FUNCTION_BLOCK Fb_CalculoCoordenadasFinalesFormacion
VAR_INPUT
	TipoCalForCavallete 					: UINT ;
	numeroLastre_int 						: UINT ;
	TipoRisultato							: UINT ;
	AlgoloAlfa_gradi						: LREAL ;
	CalculoEstacionPickinPiezasDiferentes 	: BOOL ;
	Supporto 								: POINTER TO TFMachinePalletizer_Pallet;
	XFinale 								: POINTER TO  ARRAY [1..MAXFORMINGSLAB] OF LREAL;
	
	CoorFinaleLado_Pri0_Des180 : POINTER TO ARRAY [1..MAXFORMINGSLAB] OF Es_CoordenadasCaballeteLadoA_ladoB ;
	
	YFinale 					: POINTER TO  ARRAY [1..MAXFORMINGSLAB] OF LREAL;
	YInternoLastra 				: POINTER TO  ARRAY [1..MAXFORMINGSLAB] OF LREAL;
	YCentroLastra				: POINTER TO  ARRAY [1..MAXFORMINGSLAB] OF LREAL;
	YEsternoLastra				: POINTER TO  ARRAY [1..MAXFORMINGSLAB] OF LREAL;
	YCoordinataAppoggioLastra 	: POINTER TO  ARRAY [1..MAXFORMINGSLAB] OF LREAL;
	
	ZFinale 					: POINTER TO  ARRAY [1..MAXFORMINGSLAB] OF LREAL;
	ZInternoLastra				: POINTER TO  ARRAY [1..MAXFORMINGSLAB] OF LREAL;
	ZCentroLastra      			: POINTER TO  ARRAY [1..MAXFORMINGSLAB] OF LREAL;
	ZEsternoLastra				: POINTER TO  ARRAY [1..MAXFORMINGSLAB] OF LREAL;
	
	JFinale 					: POINTER TO  ARRAY [1..MAXFORMINGSLAB] OF LREAL;
	
	XInternoLastra_A_B : POINTER TO ARRAY [1..MAXFORMINGSLAB] OF ES_SpesoreLastra_A_B;		// Coordinata X punto interno n-esima lastra depositata  (CAVALLINA-CASSA)
	YInternoLastra_A_B : POINTER TO ARRAY [1..MAXFORMINGSLAB] OF ES_SpesoreLastra_A_B;		// Coordinata Y punto interno n-esima lastra depositata  (CAVALLINA-CASSA)
	ZInternoLastra_A_B : POINTER TO ARRAY [1..MAXFORMINGSLAB] OF ES_SpesoreLastra_A_B;		// Coordinata Z punto interno n-esima lastra depositata  (CAVALLINA-CASSA)
	XCentroLastra_A_B  : POINTER TO ARRAY [1..MAXFORMINGSLAB] OF ES_SpesoreLastra_A_B;		// Coordinata X punto centrale n-esima lastra depositata  (CAVALLINA-CASSA)
	YCentroLastra_A_B  : POINTER TO ARRAY [1..MAXFORMINGSLAB] OF ES_SpesoreLastra_A_B;		// Coordinata Y punto centrale n-esima lastra depositata  (CAVALLINA-CASSA)
	ZCentroLastra_A_B  : POINTER TO ARRAY [1..MAXFORMINGSLAB] OF ES_SpesoreLastra_A_B;		// Coordinata Z punto centrale n-esima lastra depositata  (CAVALLINA-CASSA)
	XEsternoLastra_A_B : POINTER TO ARRAY [1..MAXFORMINGSLAB] OF ES_SpesoreLastra_A_B;		// Coordinata X punto esterno n-esima lastra depositata  (CAVALLINA-CASSA)
	YEsternoLastra_A_B : POINTER TO ARRAY [1..MAXFORMINGSLAB] OF ES_SpesoreLastra_A_B;		// Coordinata Y punto esterno n-esima lastra depositata  (CAVALLINA-CASSA)
	ZEsternoLastra_A_B : POINTER TO ARRAY [1..MAXFORMINGSLAB] OF ES_SpesoreLastra_A_B;		
	
	YCoordinataAppoggioLastra_A_B : POINTER TO ARRAY [1..MAXFORMINGSLAB/2] OF ES_SpesoreLastra_A_B;
	ZCoordinataAppoggioLastra_A_B : POINTER TO ARRAY [1..MAXFORMINGSLAB/2] OF ES_SpesoreLastra_A_B;
	
	
	
END_VAR
VAR_OUTPUT
END_VAR
	
VAR
	Contador						: UINT;
	varEven							: UINT;
	LadoRegistarFor					: UINT;
	NuPieza_A						: UINT;
	NuPieza_B						: UINT;
	counter2						: INT;
END_VAR


CASE TipoCalForCavallete OF
{Region "Lato DX della cavallina "}
	
	1:	// Lato DX della cavallina
		FOR Contador := 1 TO numeroLastre_int * 2 DO 
			IF NOT 	CalculoEstacionPickinPiezasDiferentes THEN 
				varEven := Contador MOD 2;
					CASE varEven OF
						0:
							XFinale^[Contador] := Supporto^.XDim/2 + Supporto^.OFSDE_X180;
							CASE TipoRisultato OF 
								0:
									XFinale^[Contador] := Supporto^.XDim/2 + Supporto^.OFSDE_X180;
									ZFinale^[Contador] := ZInternoLastra^[(Contador+varEven)/2] + Supporto^.OFSDE_Z180;
								1:
									XFinale^[Contador] := Supporto^.XDim/2 + Supporto^.OFSDE_X180;
									ZFinale^[Contador] := ZInternoLastra^[(Contador+varEven)/2] + Supporto^.OFSDE_Z180;
								3:
									XFinale^[Contador] := Supporto^.XDim/2 + Supporto^.OFSDE_X180;
									ZFinale^[Contador] := ZInternoLastra^[(Contador+varEven)/2] + Supporto^.OFSDE_Z180;
								4:
									XFinale^[Contador] := Supporto^.XDim/2 + Supporto^.OFSDE_X180;
									ZFinale^[Contador] := ZInternoLastra^[(Contador+varEven)/2] + Supporto^.OFSDE_Z180;
							END_CASE
							JFinale^[Contador] := 180 - AlgoloAlfa_gradi + Supporto^.OFSDE_J180; 
						1: 
							XFinale^[Contador] := Supporto^.XDim/2 + Supporto^.OFSDE_X0;
							CASE TipoRisultato OF 
								1:	
										
										YFinale^[Contador] := YInternoLastra^[(Contador + varEven)/2] + Supporto^.OFSDE_Y0;
										ZFinale^[Contador] := ZInternoLastra^[(Contador+varEven)/2] 	+ Supporto^.OFSDE_Z0;
									2:	
										YFinale^[Contador] := YCentroLastra^[(Contador + varEven)/2] + Supporto^.OFSDE_Y0;
										ZFinale^[Contador] := ZCentroLastra^[(Contador + varEven)/2] + Supporto^.OFSDE_Z0;
									3:	
										YFinale^[Contador] := YEsternoLastra^[(Contador + varEven)/2] + Supporto^.OFSDE_Y0;
										ZFinale^[Contador] := ZEsternoLastra^[(Contador + varEven)/2] + Supporto^.OFSDE_Z0;
									4:	
										YFinale^[Contador] := YCoordinataAppoggioLastra^[(Contador + varEven)/2] + Supporto^.OFSDE_Y0;
										ZFinale^[Contador] := ZEsternoLastra^[(Contador + varEven)/2] + Supporto^.OFSDE_Z0;
								
							END_CASE
							 JFinale^[Contador] := AlgoloAlfa_gradi + Supporto^.OFSDE_J0;
					END_CASE
			ELSIF CalculoEstacionPickinPiezasDiferentes AND Supporto^.Tipologia = CAVALLETTO THEN 
				Fun_PiezaLadoCaballete(Nu_PiezaGlobal:= Contador , Grados:= ADR(LadoRegistarFor)  ,
										 Nu_pieza_LadoA=>NuPieza_A , Nu_pieza_LadoB=> NuPieza_B  );
				CASE TipoRisultato OF 
									1:	
										CASE LadoRegistarFor OF
											0: 
												CoorFinaleLado_Pri0_Des180^[NuPieza_A].LadoA.CoordenadaFinale_X := Supporto^.XDim/2 + Supporto^.OFSDE_X0;;
												CoorFinaleLado_Pri0_Des180^[NuPieza_A].LadoA.CoordenadaFinale_Y := YInternoLastra_A_B^[NuPieza_A].Lado_A_0Grados + Supporto^.OFSDE_Y0;
												CoorFinaleLado_Pri0_Des180^[NuPieza_A].LadoA.CoordenadaFinale_Z := ZInternoLastra_A_B^[NuPieza_A].Lado_A_0Grados + Supporto^.OFSDE_Z0;
												CoorFinaleLado_Pri0_Des180^[NuPieza_A].LadoA.CoordenadaFinale_J := AlgoloAlfa_gradi + Supporto^.OFSDE_J0 ;
											180 :
												 
												CoorFinaleLado_Pri0_Des180^[NuPieza_B].LadoB.CoordenadaFinale_X := Supporto^.XDim/2 + Supporto^.OFSDE_X180;;
												CoorFinaleLado_Pri0_Des180^[NuPieza_B].LadoB.CoordenadaFinale_Y := YInternoLastra_A_B^[NuPieza_B].Lado_B_180Grados + Supporto^.OFSDE_Y0;
												CoorFinaleLado_Pri0_Des180^[NuPieza_B].LadoB.CoordenadaFinale_Z := ZInternoLastra_A_B^[NuPieza_B].Lado_B_180Grados + Supporto^.OFSDE_Z0;
												CoorFinaleLado_Pri0_Des180^[NuPieza_B].LadoB.CoordenadaFinale_J := AlgoloAlfa_gradi + Supporto^.OFSDE_J0 ;
										END_CASE
									2:	
										CASE LadoRegistarFor OF
											0: 
												CoorFinaleLado_Pri0_Des180^[NuPieza_A].LadoA.CoordenadaFinale_X := Supporto^.XDim/2 + Supporto^.OFSDE_X0;;
												CoorFinaleLado_Pri0_Des180^[NuPieza_A].LadoA.CoordenadaFinale_Y := YCentroLastra_A_B^[NuPieza_A].Lado_A_0Grados + Supporto^.OFSDE_Y0;
												CoorFinaleLado_Pri0_Des180^[NuPieza_A].LadoA.CoordenadaFinale_Z := ZCentroLastra_A_B^[NuPieza_A].Lado_A_0Grados + Supporto^.OFSDE_Z0;
												CoorFinaleLado_Pri0_Des180^[NuPieza_A].LadoA.CoordenadaFinale_J := AlgoloAlfa_gradi + Supporto^.OFSDE_J0 ;
											180 :
												 
												CoorFinaleLado_Pri0_Des180^[NuPieza_B].LadoB.CoordenadaFinale_X := Supporto^.XDim/2 + Supporto^.OFSDE_X180;;
												CoorFinaleLado_Pri0_Des180^[NuPieza_B].LadoB.CoordenadaFinale_Y := YCentroLastra_A_B^[NuPieza_B].Lado_B_180Grados + Supporto^.OFSDE_Y0;
												CoorFinaleLado_Pri0_Des180^[NuPieza_B].LadoB.CoordenadaFinale_Z := ZCentroLastra_A_B^[NuPieza_B].Lado_B_180Grados + Supporto^.OFSDE_Z0;
												CoorFinaleLado_Pri0_Des180^[NuPieza_B].LadoB.CoordenadaFinale_J := AlgoloAlfa_gradi + Supporto^.OFSDE_J0 ;
										END_CASE
									3:	
										CASE LadoRegistarFor OF
											0: 
												CoorFinaleLado_Pri0_Des180^[NuPieza_A].LadoA.CoordenadaFinale_X := Supporto^.XDim/2 + Supporto^.OFSDE_X0;;
												CoorFinaleLado_Pri0_Des180^[NuPieza_A].LadoA.CoordenadaFinale_Y := YEsternoLastra_A_B^[NuPieza_A].Lado_A_0Grados + Supporto^.OFSDE_Y0;
												CoorFinaleLado_Pri0_Des180^[NuPieza_A].LadoA.CoordenadaFinale_Z := ZEsternoLastra_A_B^[NuPieza_A].Lado_A_0Grados + Supporto^.OFSDE_Z0;
												CoorFinaleLado_Pri0_Des180^[NuPieza_A].LadoA.CoordenadaFinale_J := AlgoloAlfa_gradi + Supporto^.OFSDE_J0 ;
											180 :
												 
												CoorFinaleLado_Pri0_Des180^[NuPieza_B].LadoB.CoordenadaFinale_X := Supporto^.XDim/2 + Supporto^.OFSDE_X180;;
												CoorFinaleLado_Pri0_Des180^[NuPieza_B].LadoB.CoordenadaFinale_Y := YEsternoLastra_A_B^[NuPieza_B].Lado_B_180Grados + Supporto^.OFSDE_Y0;
												CoorFinaleLado_Pri0_Des180^[NuPieza_B].LadoB.CoordenadaFinale_Z := ZEsternoLastra_A_B^[NuPieza_B].Lado_B_180Grados + Supporto^.OFSDE_Z0;
												CoorFinaleLado_Pri0_Des180^[NuPieza_B].LadoB.CoordenadaFinale_J := AlgoloAlfa_gradi + Supporto^.OFSDE_J0 ;
										END_CASE
									4:	
										CASE LadoRegistarFor OF
											0: 
												CoorFinaleLado_Pri0_Des180^[NuPieza_A].LadoA.CoordenadaFinale_X := Supporto^.XDim/2 + Supporto^.OFSDE_X0;;
												CoorFinaleLado_Pri0_Des180^[NuPieza_A].LadoA.CoordenadaFinale_Y := YCoordinataAppoggioLastra_A_B^[NuPieza_A].Lado_A_0Grados + Supporto^.OFSDE_Y0;
												CoorFinaleLado_Pri0_Des180^[NuPieza_A].LadoA.CoordenadaFinale_Z := ZCoordinataAppoggioLastra_A_B^[NuPieza_A].Lado_A_0Grados + Supporto^.OFSDE_Z0;
												CoorFinaleLado_Pri0_Des180^[NuPieza_A].LadoA.CoordenadaFinale_J := AlgoloAlfa_gradi + Supporto^.OFSDE_J0 ;
											180 :
												 
												CoorFinaleLado_Pri0_Des180^[NuPieza_B].LadoB.CoordenadaFinale_X := Supporto^.XDim/2 + Supporto^.OFSDE_X180;;
												CoorFinaleLado_Pri0_Des180^[NuPieza_B].LadoB.CoordenadaFinale_Y := YCoordinataAppoggioLastra_A_B^[NuPieza_B].Lado_B_180Grados + Supporto^.OFSDE_Y0;
												CoorFinaleLado_Pri0_Des180^[NuPieza_B].LadoB.CoordenadaFinale_Z := ZCoordinataAppoggioLastra_A_B^[NuPieza_B].Lado_B_180Grados + Supporto^.OFSDE_Z0;
												CoorFinaleLado_Pri0_Des180^[NuPieza_B].LadoB.CoordenadaFinale_J := AlgoloAlfa_gradi + Supporto^.OFSDE_J0 ;
										END_CASE
																		
					END_CASE
							
			END_IF

	END_FOR 
{endregion}

{Region "Ordinamento consecutivo prima un lato poi l'altro"}


		(* Ordinamento consecutivo prima un lato poi l'altro *)
		2:
			FOR Contador :=1 TO numeroLastre_int BY 1 DO
				Fun_PiezaLadoCaballete(Nu_PiezaGlobal:= Contador , Grados:= ADR(LadoRegistarFor)  ,
										 Nu_pieza_LadoA=>NuPieza_A , Nu_pieza_LadoB=> NuPieza_B  );
				IF NOT CalculoEstacionPickinPiezasDiferentes THEN 
					CASE TipoRisultato OF 
							1:	
								
								CoorFinaleLado_Pri0_Des180^[Contador].LadoA.CoordenadaFinale_Y := YInternoLastra^[Contador] + Supporto^.OFSDE_Y0;
								CoorFinaleLado_Pri0_Des180^[Contador].LadoA.CoordenadaFinale_Z := ZInternoLastra^[Contador] + Supporto^.OFSDE_Z0;
								
								CoorFinaleLado_Pri0_Des180^[Contador].LadoB.CoordenadaFinale_Y := -YInternoLastra^[Contador] + Supporto^.OFSDE_Y180;
								CoorFinaleLado_Pri0_Des180^[Contador].LadoB.CoordenadaFinale_Z := ZInternoLastra^[Contador] + Supporto^.OFSDE_Z180;
								
									
	
							2:
								CoorFinaleLado_Pri0_Des180^[Contador].LadoA.CoordenadaFinale_Y := YCentroLastra^[Contador] + Supporto^.OFSDE_Y0;
								CoorFinaleLado_Pri0_Des180^[Contador].LadoA.CoordenadaFinale_Z := ZCentroLastra^[Contador] + Supporto^.OFSDE_Z0;
								
								CoorFinaleLado_Pri0_Des180^[Contador].LadoB.CoordenadaFinale_Y := -YCentroLastra^[Contador] + Supporto^.OFSDE_Y180;
								CoorFinaleLado_Pri0_Des180^[Contador].LadoB.CoordenadaFinale_Z := ZCentroLastra^[Contador] + Supporto^.OFSDE_Z180;
							
							3:
								CoorFinaleLado_Pri0_Des180^[Contador].LadoA.CoordenadaFinale_Y := YEsternoLastra^[Contador] + Supporto^.OFSDE_Y0;
								CoorFinaleLado_Pri0_Des180^[Contador].LadoA.CoordenadaFinale_Z := ZEsternoLastra^[Contador] + Supporto^.OFSDE_Z0;
								
								CoorFinaleLado_Pri0_Des180^[Contador].LadoB.CoordenadaFinale_Y := -YEsternoLastra^[Contador] + Supporto^.OFSDE_Y180;
								CoorFinaleLado_Pri0_Des180^[Contador].LadoB.CoordenadaFinale_Z := ZEsternoLastra^[Contador] + Supporto^.OFSDE_Z180;
							
							4:
								CoorFinaleLado_Pri0_Des180^[Contador].LadoA.CoordenadaFinale_Y := YCoordinataAppoggioLastra^[Contador] + Supporto^.OFSDE_Y0;
								CoorFinaleLado_Pri0_Des180^[Contador].LadoA.CoordenadaFinale_Z := ZEsternoLastra^[Contador] + Supporto^.OFSDE_Z0;
								
								CoorFinaleLado_Pri0_Des180^[Contador].LadoB.CoordenadaFinale_Y := -YCoordinataAppoggioLastra^[Contador] + Supporto^.OFSDE_Y180;
								CoorFinaleLado_Pri0_Des180^[Contador].LadoB.CoordenadaFinale_Z := ZEsternoLastra^[Contador] + Supporto^.OFSDE_Z180;
	
					END_CASE
					CoorFinaleLado_Pri0_Des180^[Contador].LadoA.CoordenadaFinale_X := Supporto^.XDim/2 + Supporto^.OFSDE_X180;
					CoorFinaleLado_Pri0_Des180^[Contador].LadoA.CoordenadaFinale_J :=  AlgoloAlfa_gradi + Supporto^.OFSDE_J0;
					CoorFinaleLado_Pri0_Des180^[Contador].LadoB.CoordenadaFinale_J := 180 - AlgoloAlfa_gradi + Supporto^.OFSDE_J180;
				ELSIF  CalculoEstacionPickinPiezasDiferentes AND Supporto^.Tipologia = CAVALLETTO  THEN 	
					
					CASE TipoRisultato OF
						1:
							CASE LadoRegistarFor OF
								0:
									CoorFinaleLado_Pri0_Des180^[NuPieza_A].LadoA.CoordenadaFinale_X := Supporto^.XDim/2 + Supporto^.OFSDE_X180;
									CoorFinaleLado_Pri0_Des180^[NuPieza_A].LadoA.CoordenadaFinale_Y := YInternoLastra_A_B^[NuPieza_A].Lado_A_0Grados + Supporto^.OFSDE_Y0;
									CoorFinaleLado_Pri0_Des180^[NuPieza_A].LadoA.CoordenadaFinale_Z := ZInternoLastra_A_B^[NuPieza_A].Lado_A_0Grados + Supporto^.OFSDE_Z0;
									CoorFinaleLado_Pri0_Des180^[NuPieza_A].LadoA.CoordenadaFinale_J := AlgoloAlfa_gradi + Supporto^.OFSDE_J0;
									
								180:
									CoorFinaleLado_Pri0_Des180^[NuPieza_B].LadoA.CoordenadaFinale_X := Supporto^.XDim/2 + Supporto^.OFSDE_X180;
									CoorFinaleLado_Pri0_Des180^[NuPieza_B].LadoB.CoordenadaFinale_Y := -YInternoLastra_A_B^[NuPieza_B].Lado_B_180Grados + Supporto^.OFSDE_Y180;
									CoorFinaleLado_Pri0_Des180^[NuPieza_B].LadoB.CoordenadaFinale_Z := ZInternoLastra_A_B^[NuPieza_B].Lado_B_180Grados + Supporto^.OFSDE_Z180;
									CoorFinaleLado_Pri0_Des180^[NuPieza_B].LadoB.CoordenadaFinale_J := 180 - AlgoloAlfa_gradi + Supporto^.OFSDE_J180;
							END_CASE
						
						
						2:
							CASE LadoRegistarFor OF
								0:
									CoorFinaleLado_Pri0_Des180^[NuPieza_A].LadoA.CoordenadaFinale_X := Supporto^.XDim/2 + Supporto^.OFSDE_X180;
									CoorFinaleLado_Pri0_Des180^[NuPieza_A].LadoA.CoordenadaFinale_Y := YCentroLastra_A_B^[NuPieza_A].Lado_A_0Grados + Supporto^.OFSDE_Y0;
									CoorFinaleLado_Pri0_Des180^[NuPieza_A].LadoA.CoordenadaFinale_Z := ZCentroLastra_A_B^[NuPieza_A].Lado_A_0Grados + Supporto^.OFSDE_Z0;
									CoorFinaleLado_Pri0_Des180^[NuPieza_A].LadoA.CoordenadaFinale_J := AlgoloAlfa_gradi + Supporto^.OFSDE_J0;
								180:
									CoorFinaleLado_Pri0_Des180^[NuPieza_B].LadoA.CoordenadaFinale_X := Supporto^.XDim/2 + Supporto^.OFSDE_X180;
									CoorFinaleLado_Pri0_Des180^[NuPieza_B].LadoB.CoordenadaFinale_Y := -YCentroLastra_A_B^[NuPieza_B].Lado_B_180Grados + Supporto^.OFSDE_Y180;
									CoorFinaleLado_Pri0_Des180^[NuPieza_B].LadoB.CoordenadaFinale_Z := ZCentroLastra_A_B^[NuPieza_B].Lado_B_180Grados + Supporto^.OFSDE_Z180;
									CoorFinaleLado_Pri0_Des180^[NuPieza_B].LadoB.CoordenadaFinale_J := 180 - AlgoloAlfa_gradi + Supporto^.OFSDE_J180;
							END_CASE
						3:
							CASE LadoRegistarFor OF
								0:
									CoorFinaleLado_Pri0_Des180^[NuPieza_A].LadoA.CoordenadaFinale_X := Supporto^.XDim/2 + Supporto^.OFSDE_X180;
									CoorFinaleLado_Pri0_Des180^[NuPieza_A].LadoA.CoordenadaFinale_Y := YEsternoLastra_A_B^[NuPieza_A].Lado_A_0Grados + Supporto^.OFSDE_Y0;
									CoorFinaleLado_Pri0_Des180^[NuPieza_A].LadoA.CoordenadaFinale_Z := ZEsternoLastra_A_B^[NuPieza_A].Lado_A_0Grados + Supporto^.OFSDE_Z0;
									CoorFinaleLado_Pri0_Des180^[NuPieza_A].LadoA.CoordenadaFinale_J := AlgoloAlfa_gradi + Supporto^.OFSDE_J0;
								180:
									CoorFinaleLado_Pri0_Des180^[NuPieza_B].LadoA.CoordenadaFinale_X := Supporto^.XDim/2 + Supporto^.OFSDE_X180;
									CoorFinaleLado_Pri0_Des180^[NuPieza_B].LadoB.CoordenadaFinale_Y := -YEsternoLastra_A_B^[NuPieza_B].Lado_B_180Grados + Supporto^.OFSDE_Y180;
									CoorFinaleLado_Pri0_Des180^[NuPieza_B].LadoB.CoordenadaFinale_Z := ZEsternoLastra_A_B^[NuPieza_B].Lado_B_180Grados + Supporto^.OFSDE_Z180;
									CoorFinaleLado_Pri0_Des180^[NuPieza_B].LadoB.CoordenadaFinale_J := 180 - AlgoloAlfa_gradi + Supporto^.OFSDE_J180;
							END_CASE
						4:
							CASE LadoRegistarFor OF
								0:
									CoorFinaleLado_Pri0_Des180^[NuPieza_A].LadoA.CoordenadaFinale_X := Supporto^.XDim/2 + Supporto^.OFSDE_X180;
									CoorFinaleLado_Pri0_Des180^[NuPieza_A].LadoA.CoordenadaFinale_Y := YCoordinataAppoggioLastra_A_B^[NuPieza_A].Lado_A_0Grados + Supporto^.OFSDE_Y0;
									CoorFinaleLado_Pri0_Des180^[NuPieza_A].LadoA.CoordenadaFinale_Z := ZEsternoLastra_A_B^[NuPieza_A].Lado_A_0Grados + Supporto^.OFSDE_Z0;
									CoorFinaleLado_Pri0_Des180^[NuPieza_A].LadoA.CoordenadaFinale_J := AlgoloAlfa_gradi + Supporto^.OFSDE_J0;
								180:
									CoorFinaleLado_Pri0_Des180^[NuPieza_B].LadoA.CoordenadaFinale_X := Supporto^.XDim/2 + Supporto^.OFSDE_X180;
									CoorFinaleLado_Pri0_Des180^[NuPieza_B].LadoB.CoordenadaFinale_Y := -YCoordinataAppoggioLastra_A_B^[NuPieza_B].Lado_B_180Grados + Supporto^.OFSDE_Y180;
									CoorFinaleLado_Pri0_Des180^[NuPieza_B].LadoB.CoordenadaFinale_Z := ZEsternoLastra_A_B^[NuPieza_B].Lado_B_180Grados + Supporto^.OFSDE_Z180;
									CoorFinaleLado_Pri0_Des180^[NuPieza_B].LadoB.CoordenadaFinale_J := 180 - AlgoloAlfa_gradi + Supporto^.OFSDE_J180;
							END_CASE
						
						
						
						
						
					END_CASE
				
				END_IF
				
				
				
				
				
				
			END_FOR
		













{endregion}
END_CASE

END_FUNCTION_BLOCK

(* stored: Version 1.1.0.1, ProductVersion 3.1.4024.11
   POU Fb_CalculoCoordenadasFinalesFormacion: Id {a2b34fcb-80d8-4f40-83a2-c1979dfcf9f9}, SpecialFunc None *)
